Omron Sysmac Studio project ModbuTCP_Test_Project_v2 (Sysmac Studio 1.47.0.64008, StandardProject)

# Controller new_Controller_0: NX102-1220 version 1.38
Task PrimaryTask (priority 4, period or condition 2000): Program0

TYPE DUT_srtBasic : STRUCT
    Busy : BOOL;
    Error : BOOL;
    ErrorID : WORD;
    Done : BOOL;
END_STRUCT END_TYPE
TYPE DUT_ModbusTCPReadStatus : STRUCT
    Basic : DUT_srtBasic;
    ErrorIDEx : DWORD;
    ReadSize : UINT;
END_STRUCT END_TYPE

PROGRAM Program0
VAR
    _SktTCPConnect : SktTCPConnect;
    _SktTCPClose : SktClose;
    bExecute : BOOL;
    bClose : BOOL;
    Socket : _sSOCKET;
    _ModbusTCPRead : ModbusTCPRead;
    _ModbusTCPReadCoils : ModbusTCPRead;
    bError : BOOL;
    ModbusReadDat : ARRAY[0..99] OF word;
    ModbusWriteDat : ARRAY[0..99] OF word;
    ModbusReadDataCoils : ARRAY[0..99] OF bool;
    ModbusWrite_16 : ARRAY[0..99] OF word;  (* Pilz:ModbusRegister04_Read *)
    ModbusRead_03 : ARRAY[0..99] OF word;  (* Pilz:ModbusRegister03_Write *)
    ModbusRead_04 : ARRAY[0..99] OF word;  (* Pilz:ModbusRegister04_Write *)
    ModbusRead_01 : ARRAY[0..99] OF bool;  (* Pilz:ModbusCoil00_Write *)
    ModbusRead_02 : ARRAY[0..99] OF bool;  (* Pilz:ModbusCoil01_Write *)
    ModbusWrite_15 : ARRAY[0..99] OF bool;  (* Pilz:ModbusCoil00_Read *)
    ReadCmd : _sMODBUS_READ;
    bReads : ARRAY[0..15] OF bool;
    iStep : INT;
    bWrites : ARRAY[0..15] OF bool;
    bStart : BOOL;
    R_TRIG1 : R_TRIG;  (* Start Edge *)
    ModbusTCPReadStatus : DUT_ModbusTCPReadStatus;
    ModbusTCPReadCoilStatus : DUT_ModbusTCPReadStatus;
    SktBasicStatus : DUT_srtBasic;  (* Socket Connect FB Status *)
    SktCloseStatus : DUT_srtBasic;  (* Socket Close FB Status *)
    _SktSetOption : SktSetOption;
    SktSetOptionStatus : DUT_srtBasic;
    bSetOptions : BOOL;
    bOptionNoDelay : BOOL := True;
    TONs : ARRAY[0..15] OF ton;
    Dummy : BOOL;
    _ModbusTCPWriteRegister : ModbusTCPWrite;
    WriteCmd : _sMODBUS_WRITE;
    ModbusTCPWriteRegisterStatus : DUT_ModbusTCPReadStatus;
    ModbusWriteDatCoils : ARRAY[0..99] OF bool;
    _ModbusTCPWriteCoils : ModbusTCPWrite;
    ModbusTCPWriteCoilsStatus : DUT_ModbusTCPReadStatus;
END_VAR
VAR
    _p1 : BOOL;
    _p2 : BOOL;
    _t3 : BOOL;
    _p4 : BOOL;
    _t5 : BOOL;
    _p6 : BOOL;
    _t7 : BOOL;
    _p8 : BOOL;
    _t9 : BOOL;
    _p10 : BOOL;
    _t11 : BOOL;
    _p12 : BOOL;
    _t13 : BOOL;
    _p14 : BOOL;
    _p15 : BOOL;
END_VAR

(* Section Section0: ladder, written here as Structured Text *)

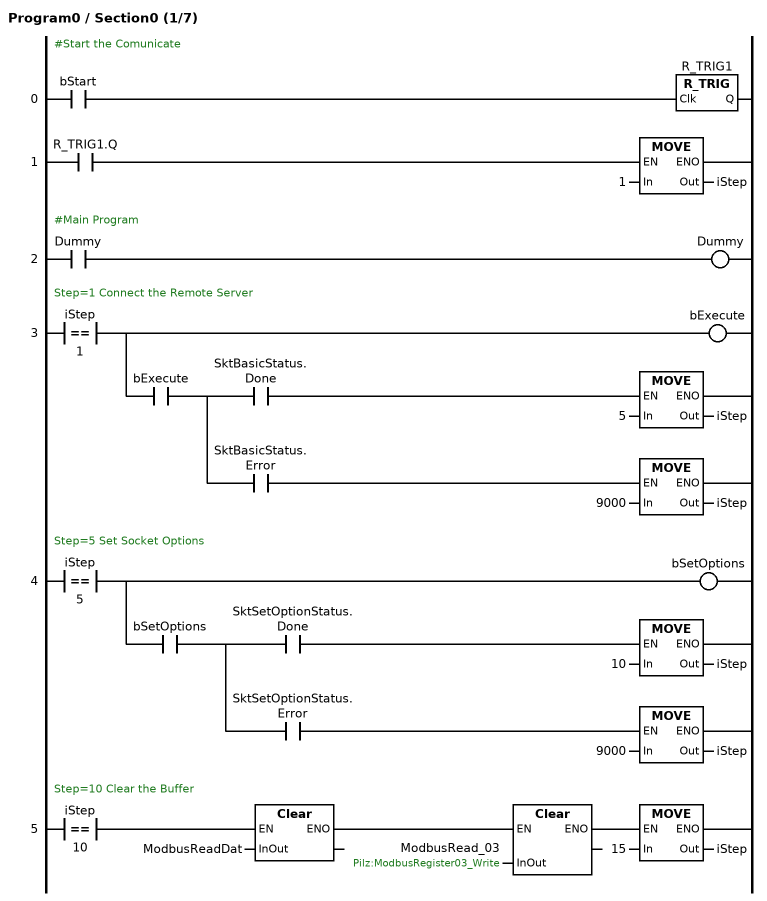
(* Rung 0: #Start the Comunicate *)
R_TRIG1(Clk := bStart);
(* Rung 1 *)
IF R_TRIG1.Q THEN iStep := 1; END_IF;
(* Rung 2: #Main Program *)
Dummy := Dummy;
(* Rung 3: Step=1 Connect the Remote Server *)
bExecute := iStep = 1;
_p1 := (iStep = 1) AND bExecute;
IF (iStep = 1) AND bExecute AND SktBasicStatus.Done THEN iStep := 5; END_IF;
IF _p1 AND SktBasicStatus.Error THEN iStep := 9000; END_IF;
(* Rung 4: Step=5 Set Socket Options *)
bSetOptions := iStep = 5;
_p2 := (iStep = 5) AND bSetOptions;
IF (iStep = 5) AND bSetOptions AND SktSetOptionStatus.Done THEN iStep := 10; END_IF;
IF _p2 AND SktSetOptionStatus.Error THEN iStep := 9000; END_IF;
(* Rung 5: Step=10 Clear the Buffer *)
IF iStep = 10 THEN
    Clear(InOut := ModbusReadDat);
    Clear(InOut := ModbusRead_03);
    iStep := 15;
END_IF;

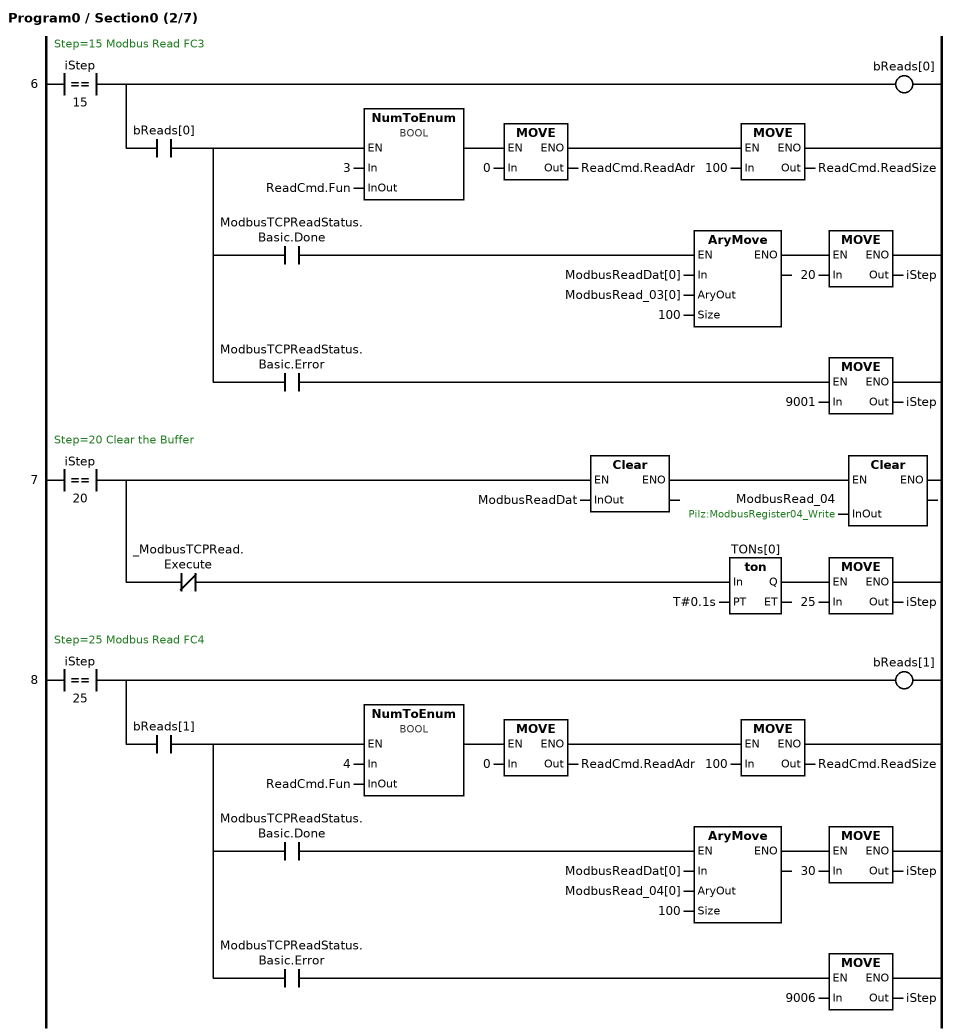
(* Rung 6: Step=15 Modbus Read FC3 *)
bReads[0] := iStep = 15;
_t3 := FALSE;
IF (iStep = 15) AND bReads[0] THEN _t3 := NumToEnum(In := 3, InOut := ReadCmd.Fun); END_IF;
IF _t3 THEN
    ReadCmd.ReadAdr := 0;
    ReadCmd.ReadSize := 100;
END_IF;
IF (iStep = 15) AND bReads[0] AND ModbusTCPReadStatus.Basic.Done THEN
    AryMove(In := ModbusReadDat[0], AryOut := ModbusRead_03[0], Size := 100);
END_IF;
_p4 := (iStep = 15) AND bReads[0];
IF (iStep = 15) AND bReads[0] AND ModbusTCPReadStatus.Basic.Done THEN iStep := 20; END_IF;
IF _p4 AND ModbusTCPReadStatus.Basic.Error THEN iStep := 9001; END_IF;
(* Rung 7: Step=20 Clear the Buffer *)
IF iStep = 20 THEN
    Clear(InOut := ModbusReadDat);
    Clear(InOut := ModbusRead_04);
END_IF;
TONs[0](In := (iStep = 20) AND NOT _ModbusTCPRead.Execute, PT := T#0.1s);
IF TONs[0].Q THEN iStep := 25; END_IF;
(* Rung 8: Step=25 Modbus Read FC4 *)
bReads[1] := iStep = 25;
_t5 := FALSE;
IF (iStep = 25) AND bReads[1] THEN _t5 := NumToEnum(In := 4, InOut := ReadCmd.Fun); END_IF;
IF _t5 THEN
    ReadCmd.ReadAdr := 0;
    ReadCmd.ReadSize := 100;
END_IF;
IF (iStep = 25) AND bReads[1] AND ModbusTCPReadStatus.Basic.Done THEN
    AryMove(In := ModbusReadDat[0], AryOut := ModbusRead_04[0], Size := 100);
END_IF;
_p6 := (iStep = 25) AND bReads[1];
IF (iStep = 25) AND bReads[1] AND ModbusTCPReadStatus.Basic.Done THEN iStep := 30; END_IF;
IF _p6 AND ModbusTCPReadStatus.Basic.Error THEN iStep := 9006; END_IF;

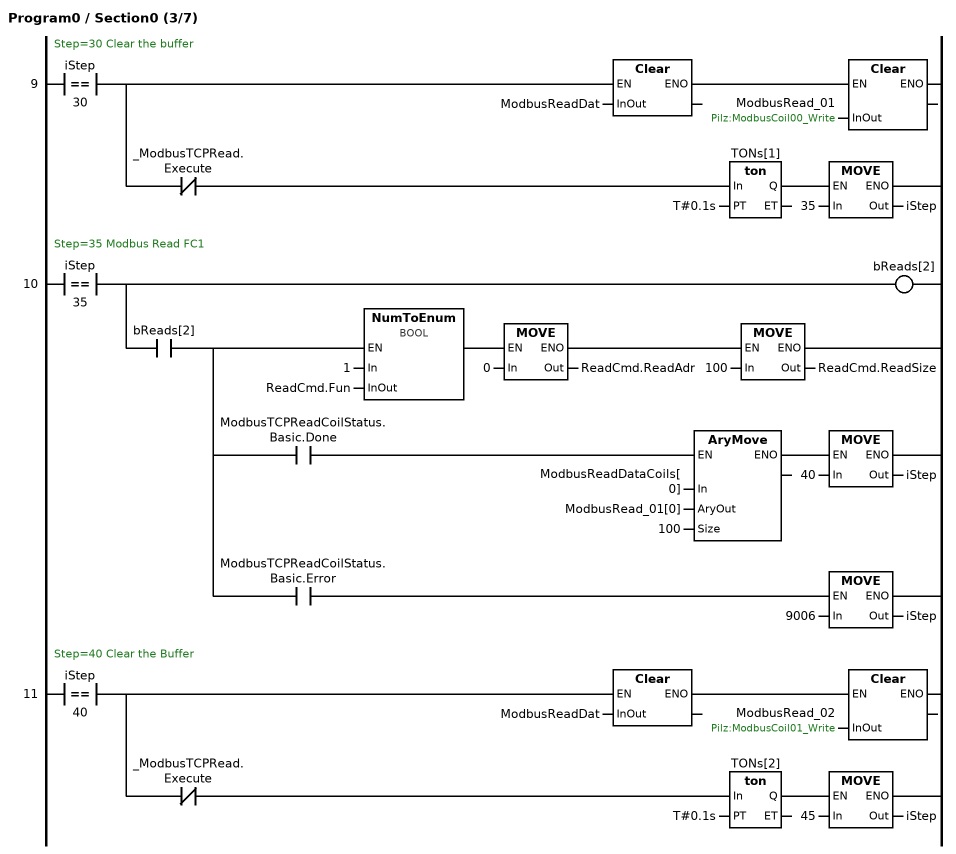
(* Rung 9: Step=30 Clear the buffer *)
IF iStep = 30 THEN
    Clear(InOut := ModbusReadDat);
    Clear(InOut := ModbusRead_01);
END_IF;
TONs[1](In := (iStep = 30) AND NOT _ModbusTCPRead.Execute, PT := T#0.1s);
IF TONs[1].Q THEN iStep := 35; END_IF;
(* Rung 10: Step=35 Modbus Read FC1 *)
bReads[2] := iStep = 35;
_t7 := FALSE;
IF (iStep = 35) AND bReads[2] THEN _t7 := NumToEnum(In := 1, InOut := ReadCmd.Fun); END_IF;
IF _t7 THEN
    ReadCmd.ReadAdr := 0;
    ReadCmd.ReadSize := 100;
END_IF;
IF (iStep = 35) AND bReads[2] AND ModbusTCPReadCoilStatus.Basic.Done THEN
    AryMove(In := ModbusReadDataCoils[0], AryOut := ModbusRead_01[0], Size := 100);
END_IF;
_p8 := (iStep = 35) AND bReads[2];
IF (iStep = 35) AND bReads[2] AND ModbusTCPReadCoilStatus.Basic.Done THEN iStep := 40; END_IF;
IF _p8 AND ModbusTCPReadCoilStatus.Basic.Error THEN iStep := 9006; END_IF;
(* Rung 11: Step=40 Clear the Buffer *)
IF iStep = 40 THEN
    Clear(InOut := ModbusReadDat);
    Clear(InOut := ModbusRead_02);
END_IF;
TONs[2](In := (iStep = 40) AND NOT _ModbusTCPRead.Execute, PT := T#0.1s);
IF TONs[2].Q THEN iStep := 45; END_IF;

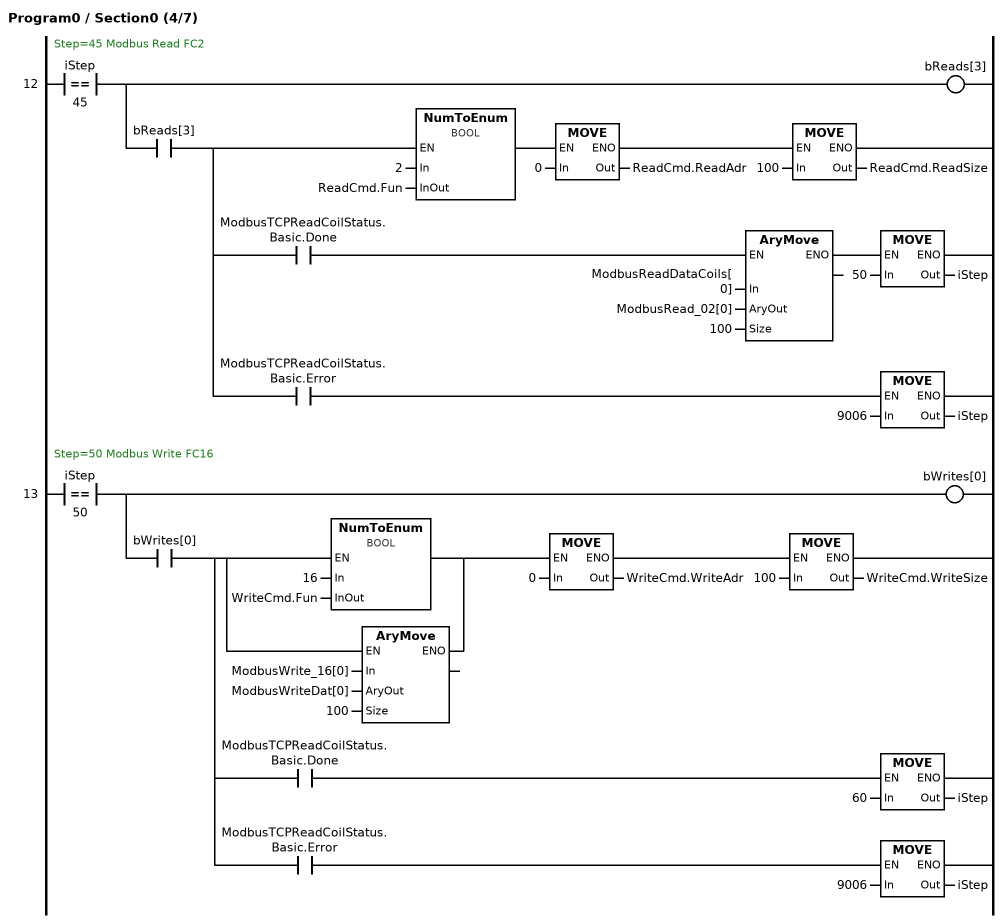
(* Rung 12: Step=45 Modbus Read FC2 *)
bReads[3] := iStep = 45;
_t9 := FALSE;
IF (iStep = 45) AND bReads[3] THEN _t9 := NumToEnum(In := 2, InOut := ReadCmd.Fun); END_IF;
IF _t9 THEN
    ReadCmd.ReadAdr := 0;
    ReadCmd.ReadSize := 100;
END_IF;
IF (iStep = 45) AND bReads[3] AND ModbusTCPReadCoilStatus.Basic.Done THEN
    AryMove(In := ModbusReadDataCoils[0], AryOut := ModbusRead_02[0], Size := 100);
END_IF;
_p10 := (iStep = 45) AND bReads[3];
IF (iStep = 45) AND bReads[3] AND ModbusTCPReadCoilStatus.Basic.Done THEN iStep := 50; END_IF;
IF _p10 AND ModbusTCPReadCoilStatus.Basic.Error THEN iStep := 9006; END_IF;
(* Rung 13: Step=50 Modbus Write FC16 *)
bWrites[0] := iStep = 50;
_t11 := FALSE;
IF (iStep = 50) AND bWrites[0] THEN _t11 := NumToEnum(In := 16, InOut := WriteCmd.Fun); END_IF;
IF (iStep = 50) AND bWrites[0] THEN
    AryMove(In := ModbusWrite_16[0], AryOut := ModbusWriteDat[0], Size := 100);
END_IF;
IF _t11 OR ((iStep = 50) AND bWrites[0]) THEN
    WriteCmd.WriteAdr := 0;
    WriteCmd.WriteSize := 100;
END_IF;
_p12 := (iStep = 50) AND bWrites[0];
IF (iStep = 50) AND bWrites[0] AND ModbusTCPReadCoilStatus.Basic.Done THEN iStep := 60; END_IF;
IF _p12 AND ModbusTCPReadCoilStatus.Basic.Error THEN iStep := 9006; END_IF;

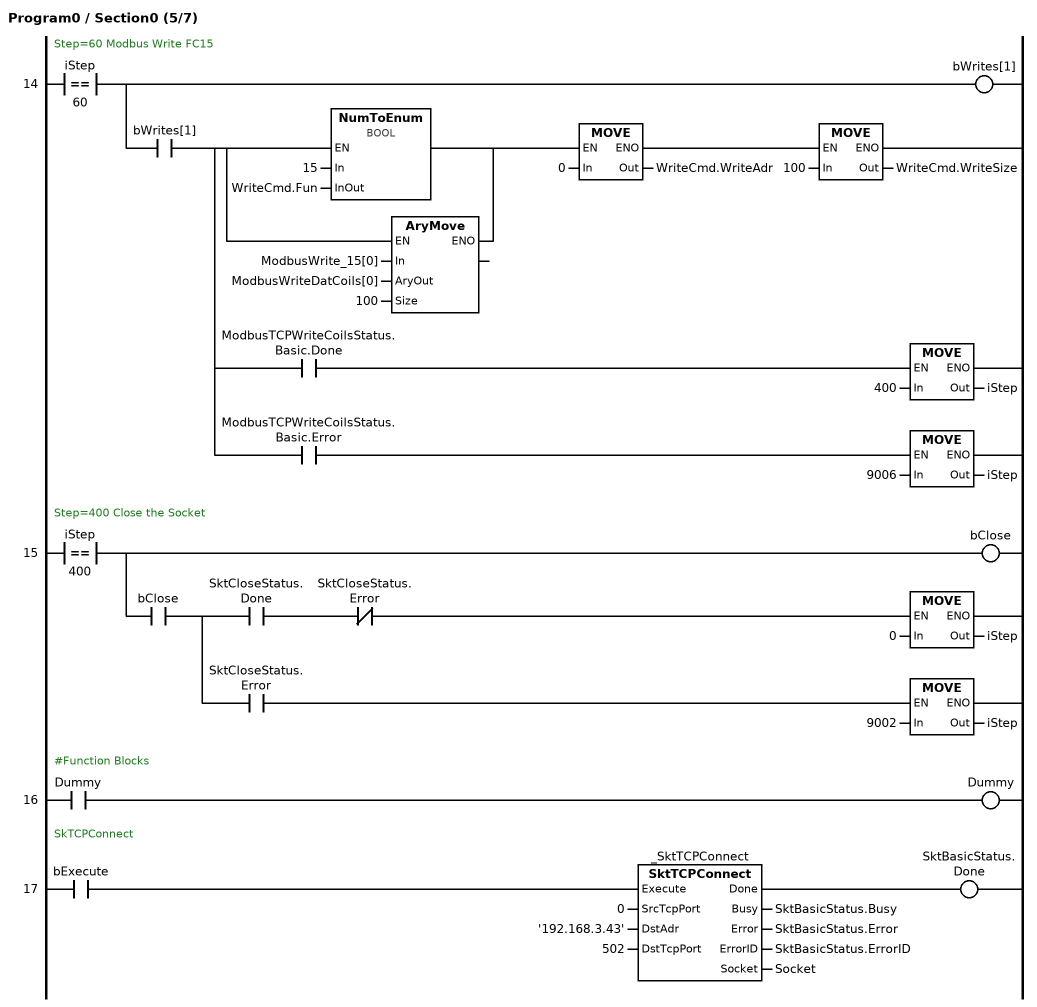
(* Rung 14: Step=60 Modbus Write FC15 *)
bWrites[1] := iStep = 60;
_t13 := FALSE;
IF (iStep = 60) AND bWrites[1] THEN _t13 := NumToEnum(In := 15, InOut := WriteCmd.Fun); END_IF;
IF (iStep = 60) AND bWrites[1] THEN
    AryMove(In := ModbusWrite_15[0], AryOut := ModbusWriteDatCoils[0], Size := 100);
END_IF;
IF _t13 OR ((iStep = 60) AND bWrites[1]) THEN
    WriteCmd.WriteAdr := 0;
    WriteCmd.WriteSize := 100;
END_IF;
_p14 := (iStep = 60) AND bWrites[1];
IF (iStep = 60) AND bWrites[1] AND ModbusTCPWriteCoilsStatus.Basic.Done THEN iStep := 400; END_IF;
IF _p14 AND ModbusTCPWriteCoilsStatus.Basic.Error THEN iStep := 9006; END_IF;
(* Rung 15: Step=400 Close the Socket *)
bClose := iStep = 400;
_p15 := (iStep = 400) AND bClose;
IF (iStep = 400) AND bClose AND SktCloseStatus.Done AND NOT SktCloseStatus.Error THEN iStep := 0; END_IF;
IF _p15 AND SktCloseStatus.Error THEN iStep := 9002; END_IF;
(* Rung 16: #Function Blocks *)
Dummy := Dummy;
(* Rung 17: SkTCPConnect *)
_SktTCPConnect(Execute := bExecute, SrcTcpPort := 0, DstAdr := '192.168.3.43', DstTcpPort := 502, Busy => SktBasicStatus.Busy, Error => SktBasicStatus.Error, ErrorID => SktBasicStatus.ErrorID, Socket => Socket);
SktBasicStatus.Done := _SktTCPConnect.Done;

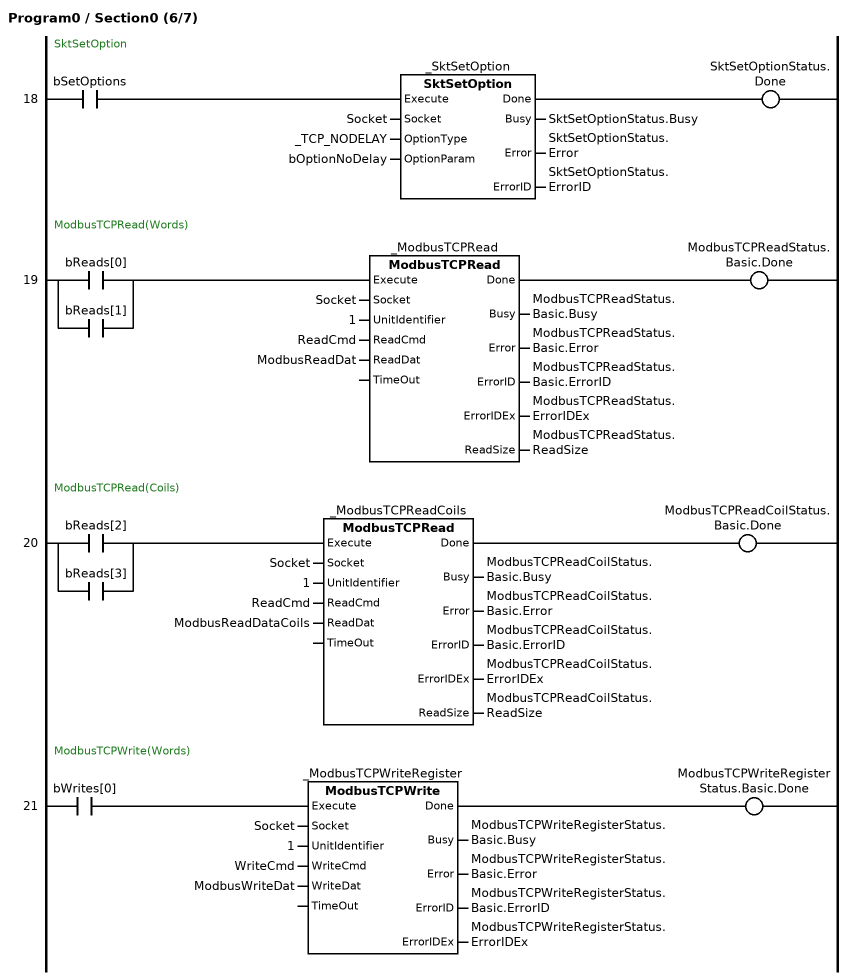
(* Rung 18: SktSetOption *)
_SktSetOption(Execute := bSetOptions, Socket := Socket, OptionType := _TCP_NODELAY, OptionParam := bOptionNoDelay, Busy => SktSetOptionStatus.Busy, Error => SktSetOptionStatus.Error, ErrorID => SktSetOptionStatus.ErrorID);
SktSetOptionStatus.Done := _SktSetOption.Done;
(* Rung 19: ModbusTCPRead(Words) *)
_ModbusTCPRead(Execute := bReads[0] OR bReads[1], Socket := Socket, UnitIdentifier := 1, ReadCmd := ReadCmd, ReadDat := ModbusReadDat, Busy => ModbusTCPReadStatus.Basic.Busy, Error => ModbusTCPReadStatus.Basic.Error, ErrorID => ModbusTCPReadStatus.Basic.ErrorID, ErrorIDEx => ModbusTCPReadStatus.ErrorIDEx, ReadSize => ModbusTCPReadStatus.ReadSize);
ModbusTCPReadStatus.Basic.Done := _ModbusTCPRead.Done;
(* Rung 20: ModbusTCPRead(Coils) *)
_ModbusTCPReadCoils(Execute := bReads[2] OR bReads[3], Socket := Socket, UnitIdentifier := 1, ReadCmd := ReadCmd, ReadDat := ModbusReadDataCoils, Busy => ModbusTCPReadCoilStatus.Basic.Busy, Error => ModbusTCPReadCoilStatus.Basic.Error, ErrorID => ModbusTCPReadCoilStatus.Basic.ErrorID, ErrorIDEx => ModbusTCPReadCoilStatus.ErrorIDEx, ReadSize => ModbusTCPReadCoilStatus.ReadSize);
ModbusTCPReadCoilStatus.Basic.Done := _ModbusTCPReadCoils.Done;
(* Rung 21: ModbusTCPWrite(Words) *)
_ModbusTCPWriteRegister(Execute := bWrites[0], Socket := Socket, UnitIdentifier := 1, WriteCmd := WriteCmd, WriteDat := ModbusWriteDat, Busy => ModbusTCPWriteRegisterStatus.Basic.Busy, Error => ModbusTCPWriteRegisterStatus.Basic.Error, ErrorID => ModbusTCPWriteRegisterStatus.Basic.ErrorID, ErrorIDEx => ModbusTCPWriteRegisterStatus.ErrorIDEx);
ModbusTCPWriteRegisterStatus.Basic.Done := _ModbusTCPWriteRegister.Done;

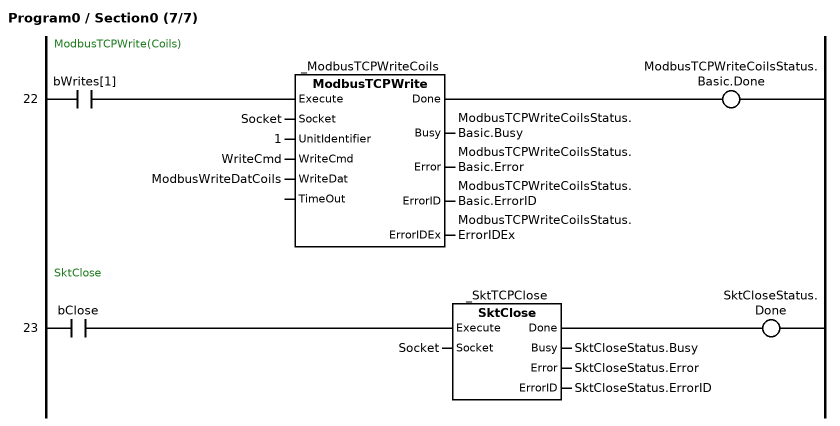
(* Rung 22: ModbusTCPWrite(Coils) *)
_ModbusTCPWriteCoils(Execute := bWrites[1], Socket := Socket, UnitIdentifier := 1, WriteCmd := WriteCmd, WriteDat := ModbusWriteDatCoils, Busy => ModbusTCPWriteCoilsStatus.Basic.Busy, Error => ModbusTCPWriteCoilsStatus.Basic.Error, ErrorID => ModbusTCPWriteCoilsStatus.Basic.ErrorID, ErrorIDEx => ModbusTCPWriteCoilsStatus.ErrorIDEx);
ModbusTCPWriteCoilsStatus.Basic.Done := _ModbusTCPWriteCoils.Done;
(* Rung 23: SktClose *)
_SktTCPClose(Execute := bClose, Socket := Socket, Busy => SktCloseStatus.Busy, Error => SktCloseStatus.Error, ErrorID => SktCloseStatus.ErrorID);
SktCloseStatus.Done := _SktTCPClose.Done;
END_PROGRAM